INTERFACE I_ActuatorEnableDisable EXTENDS I_ActuatorBase

{attribute 'monitoring' := 'call'}
PROPERTY public isDisabled : BOOL
GET
END_GET
END_PROPERTY

{attribute 'monitoring' := 'call'}
PROPERTY public isEnabled : BOOL
GET
END_GET
END_PROPERTY

METHOD public setDisable : BOOL
VAR_INPUT
END_VAR
END_METHOD

METHOD public setEnable : BOOL
VAR_INPUT
END_VAR
END_METHOD

END_INTERFACE

(* stored: Version 1.1.0.1, ProductVersion 3.1.4024.3
   Itf I_ActuatorEnableDisable: Id {5129998d-d586-4aab-ae89-8f8159dfea5a}
   Property isDisabled: Id {5617a1b0-d471-4fc4-9ecb-6f6c3c9b6dd9}
   Get Get: Id {14facebd-60e7-43be-93b2-ffbde5517ab9}
   Property isEnabled: Id {24157986-6f8d-4387-ba9f-9dc726bd9e62}
   Get Get: Id {93943023-dcbe-4c64-bcc8-6578590e63b4}
   Method setDisable: Id {655253f9-38a5-410e-9595-a86e54d5afe9}
   Method setEnable: Id {008bd135-b8c7-4057-aea8-2b642a5b5247} *)
